(* IEC 61131-3 sources: JaccoSigma/tempclass/Class/ET_User, 1 file *)

(* ---- ET_User.st ---- *)
(*!
<Class
	Name               = "ET_User"
	Revision           = "1.0"
	RealtimeTask       = "false"
	CyclicTask         = "false"
	BackgroundTask     = "false"
	Sigmatek           = "true"
	OSInterface        = "false"
	HighPriority       = "false"
	Automatic          = "false"
	UpdateMode         = "Prescan"
	IconPath           = ".\Class\ET_User\toolbox.ICO"
	SharedCommandTable = "true"
	Objectsize         = "(284,120)"
	Comment            = "V1.0&#13;&#10;Class for user functions, called by LasalText">
	<Channels>
		<Server Name="Server0" Visualized="true" Initialize="false" WriteProtected="false" Retentive="false" Comment="connect to Client User of _ET_Runtime "/>
	</Channels>
</Class>
*)
ET_User : CLASS
  //Servers:
	Server0 	: SvrChCmd_DINT;
  //Clients:
  //Variables:
  //Functions:
				//! <Function Comment="Userfunction called by LasalText" Name="FC_User"/>
	FUNCTION VIRTUAL GLOBAL FC_User
		VAR_INPUT
			no 	: DINT;			//! <Variable Comment="number...     if there is more than on user function&#13;&#10;" Name="FC_User.no"/>
			parameter 	: DINT;			//! <Variable Comment="parameter...  the parameter for the function" Name="FC_User.parameter"/>
		END_VAR;
  //Tables:
	FUNCTION @STD
		VAR_OUTPUT
			ret_code	: CONFSTATES;
		END_VAR;
	FUNCTION GLOBAL TAB @CT_;
END_CLASS;

//*********************Inserted from .\ET_User\ET_User_00_00.st*********************

FUNCTION VIRTUAL GLOBAL ET_User::FC_User
VAR_INPUT
	no		: DINT;
	parameter		: DINT;
END_VAR
VAR
    para    : DINT;
END_VAR;

  para := parameter;
  case no of
	   1:
	   2:
       3:
  end_case;

END_FUNCTION //GLOBAL ET_User::FC_User
